// TIA Portal V20 export
TYPE "LER_typeAxisCommand"
// stored: Access Published
   STRUCT
      general : Bool;
      jogForward : Bool;
      jogBackward : Bool;
      moveVelocity : Bool;
      torqueLimiting : Bool;
      homing : Bool;
      posRelative : Bool;
      posAbsoluteSummary : Bool;
      posAbsolute : Array[0..15] of Bool;
   END_STRUCT;
END_TYPE
